PROGRAM MAIN
VAR
	fbXml					: FB_XmlDomParser;
	
	xmlDoc					: SXmlNode;

	xmlMachines				: SXmlNode;
	xmlMachine1				: SXmlNode;
	xmlMachine2				: SXmlNode;
	
	xmlIterator				: SXmlIterator;
	xmlMachineNode			: SXmlNode;
	xmlMachineNodeValue		: STRING;		
	
	xmlMachine1Attribute	: SXmlAttribute;
	xmlMachine2Attribute	: SXmlAttribute;
	
	sMachine1Name			: STRING;
	sMachine2Name			: STRING;
	
	nMachine1Attribute		: DINT;
	nMachine2Attribute		: DINT;
	
	sMessageToParse			: STRING(255) := '<Machines><Machine Type="1">Wilde Nelli</Machine><Machine Type="2">Huber8</Machine></Machines>';
	
	i : INT;
END_VAR

(* Load XML content *)
xmlDoc := fbXml.ParseDocument(sMessageToParse);

(* Parse XML nodes - Option 1 *)
xmlMachines := fbXml.ChildByName(xmlDoc, 'Machines');
xmlMachine1 := fbXml.ChildByAttribute(xmlMachines, 'Type', '1');
xmlMachine2 := fbXml.ChildByAttributeAndName(xmlMachines, 'Type', '2', 'Machine');

(* Parse XML nodes - Option 2 *)
xmlMachines := fbXml.ChildByName(xmlDoc, 'Machines');
xmlMachineNode := fbXml.ChildrenByName(xmlMachines, xmlIterator, 'Machine');
WHILE NOT fbXml.IsEnd(xmlIterator) DO
	xmlMachineNode := fbXml.Node(xmlIterator);
	xmlMachineNodeValue := fbXml.NodeText(xmlMachineNode);
	XmlIterator := fbXml.Next(XmlIterator);
END_WHILE

(* Parse XML attributes *)
xmlMachine1Attribute := fbXml.Attribute(xmlMachine1, 'Type');
xmlMachine2Attribute := fbXml.Attribute(xmlMachine2, 'Type');

(* Retrieve node values *)
sMachine1Name := fbXml.NodeText(xmlMachine1);
sMachine2Name := fbXml.NodeText(xmlMachine2);

(* Retrieve attribute values *)
nMachine1Attribute := fbXml.AttributeAsInt(xmlMachine1Attribute);
nMachine2Attribute := fbXml.AttributeAsInt(xmlMachine2Attribute);

END_PROGRAM

(* stored: Version 1.1.0.1, ProductVersion 3.1.4022.12
   POU MAIN: Id {ed120519-6aa8-4fd0-87ed-ffa0c7751332}, SpecialFunc None *)
